TYPE "Station information_ShW"
VERSION : 0.1
   STRUCT
      TowerLampStatus : Int;
      "SafetyDoor Trigger" : Bool;
      "EmergencyStop Trigger" : Bool;
      StationMode : Int;
      StationStatus : Int;
      SubStationCycleRunning : Bool;
   END_STRUCT;

END_TYPE

